// TIA Portal V18 export
TYPE "UDT_LabelFeeder"
// stored: IsFailsafeCompliant false
   STRUCT
      Manual : Struct
         Star : Bool;
         Rest : Bool;
      END_STRUCT;
      Auto : Struct
         Star : Bool;
         Rest : Bool;
      END_STRUCT;
      In : Struct
         ReadyOK : Bool;
         ALM : Bool;
      END_STRUCT;
      Out : Struct
         Star : Bool;
         Rest : Bool;
      END_STRUCT;
   END_STRUCT;
END_TYPE
